FUNCTION_BLOCK Test_TStreamAdd_Read_STRING EXTENDS TUnitTestBase
VAR
    Stream : TStream(StreamLength := 2);
    TestString : STRING := '111111111 222222222 333333333 444444444 555555555 666666666 777777777 888888888 ';
END_VAR



Stream.Init(2);

Stream.Add_STRING(TestString);
    
Assertion.AssertEquals_UDINT(
    Expected := 81,
    Actual := Stream.Position,
    ObjectName := _TestName,
    VariableName := 'Stream.Position');
    
Stream.Seek(0);

Assertion.AssertEquals_STRING(
    Expected := TestString,
    Actual := Stream.Read_STRING(),
    ObjectName := _TestName,
    VariableName := 'Stream.Read_STRING()');
    
Assertion.AssertEquals_UDINT(
    Expected := 81,
    Actual := Stream.Position,
    ObjectName := _TestName,
    VariableName := 'Stream.Position');
    
    
TestFinished();

END_FUNCTION_BLOCK

(* stored: Version 1.1.0.1, ProductVersion 3.1.4024.4
   POU Test_TStreamAdd_Read_STRING: Id {71d42138-05d4-455e-ad1d-63fac6ca418e}, SpecialFunc None *)
